FUNCTION_BLOCK FB_AnalogInputScalingPlusMinus
VAR_INPUT
	nRawInput 				: INT;
	stAnalogInputScaling    : ST_AnalogInputScaling_1;
END_VAR
VAR_OUTPUT
	fOutput 				: LREAL;
END_VAR
VAR
	fRawInput 				: LREAL;
	fNormalizedInput		: LREAL;
END_VAR

fRawInput := INT_TO_LREAL(nRawInput);

fNormalizedInput := (stAnalogInputScaling.fMaxOutputValue - stAnalogInputScaling.fMinOutputValue)/2 + (fRawInput/stAnalogInputScaling.fMaxInputValue)*((stAnalogInputScaling.fMaxOutputValue - stAnalogInputScaling.fMinOutputValue)/2);

fOutput := LIMIT(stAnalogInputScaling.fMinOutputValue, fNormalizedInput, stAnalogInputScaling.fMaxOutputValue);

//fNormalizedInput := (fRawInput - stAnalogInputScaling.fMinInputValue) / (stAnalogInputScaling.fMaxInputValue - stAnalogInputScaling.fMinInputValue);

//fOutput := LIMIT(stAnalogInputScaling.fMinOutputValue, stAnalogInputScaling.fMinOutputValue + fNormalizedInput*(stAnalogInputScaling.fMaxOutputValue - stAnalogInputScaling.fMinOutputValue), stAnalogInputScaling.fMaxOutputValue);

END_FUNCTION_BLOCK

(* stored: Version 1.1.0.1, ProductVersion 3.1.4024.12
   POU FB_AnalogInputScalingPlusMinus: Id {b792c456-0f10-462e-b521-73238f1621f3}, SpecialFunc None *)
